// TIA Portal V19 export
TYPE "FeedMachine_Alr"
// stored: Access Published
   STRUCT
      BrakeTimeOut { S7_SetPoint := 'True'} : Bool;
      Ax : "TAx_Speed_Alarms";
      Fan_M { S7_SetPoint := 'True'} : "MotorAlr";
   END_STRUCT;
END_TYPE
